PROGRAM P31_PriorityControl
VAR
	fbAnalogDeviceRampControl : FB_AnalogDeviceRampControl;
	pr_TON: TON;
END_VAR
VAR_OUTPUT
	complete : BOOL;
END_VAR

pr_TON(IN := TRUE, PT := (1 + GVL_INTERFACE_UI.aAnalogController[1].cvController.input.rampTime) * T#1S);
fbAnalogDeviceRampControl();
IF pr_TON.Q = TRUE THEN
	pr_TON(IN := FALSE);
	complete := TRUE;
ELSE 
	complete := FALSE;
END_IF

END_PROGRAM

(* stored: Version 1.1.0.1, ProductVersion 3.1.4026.11
   POU P31_PriorityControl: Id {1b30a652-8bf4-4fa2-bbbd-1c67b04f4c5a}, SpecialFunc None *)
